// 隐含生成代码：不要编辑
FUNCTION CheckRangeUnsigned : UDINT
VAR_INPUT
	value, lower, upper: UDINT;
END_VAR

// 隐含生成代码：这里只是对代码实现的建议
{noflow}
IF (value < lower) THEN
	CheckRangeUnsigned := lower;
ELSIF(value > upper) THEN
	CheckRangeUnsigned := upper;
ELSE
	CheckRangeUnsigned := value;
END_IF
{flow}

END_FUNCTION

(* stored: Version 1.1.0.1, ProductVersion 3.1.4022.16
   POU CheckRangeUnsigned: Id {cf2b4250-d1d5-423b-b72d-249dae848a6e}, SpecialFunc CheckRangeUnsigned *)
